{attribute 'linkalways'} 
{attribute 'no_explicit_call' := 'This FB is a CLASS and must be accessed using methods or properties'}
{attribute 'enable_dynamic_creation'}
FUNCTION_BLOCK Node_F_VN_GetPerspectiveTransformation EXTENDS VisionNode
VAR
	aSrcPoints : _TcVnArray4_Point2_REAL;
    aDestPoints : _TcVnArray4_Point2_REAL;
    aTransformationMatrix : _TcVnMatrix3x3_LREAL;
    hrPrev : _HRESULT(S_OK);
	hresult : _HRESULT(S_OK);
END_VAR

METHOD PUBLIC  Clone : I_Node
VAR
	pNode : POINTER TO Node_F_VN_GetPerspectiveTransformation;
END_VAR
pNode := __NEW(Node_F_VN_GetPerspectiveTransformation);
Clone := pNode^;
END_METHOD

METHOD FB_init : BOOL
VAR_INPUT
	bInitRetains : BOOL; // if TRUE, the retain variables are initialized (warm start / cold start)
	bInCopyCode : BOOL;  // if TRUE, the instance afterwards gets moved into the copy code (online change)
END_VAR
AddInput('aSrcPoints', aSrcPoints);
AddInput('aDestPoints', aDestPoints);
AddInput('hrPrev', hrPrev);
AddOutput('aTransformationMatrix', aTransformationMatrix);
AddOutput('hresult',hresult);
END_METHOD

METHOD PROTECTED OnExecute
hresult.Value := F_VN_GetPerspectiveTransformation(
	aSrcPoints := aSrcPoints.Value, 
	aDestPoints := aDestPoints.Value, 
	aTransformationMatrix := aTransformationMatrix.Value, 
	hrPrev := hrPrev.Value);
END_METHOD

METHOD PUBLIC PreExecutionCheck
VAR_INPUT
	Check : I_PreExecutionChecks;
END_VAR
END_METHOD

END_FUNCTION_BLOCK

(* stored: Version 1.1.0.1, ProductVersion 3.1.4024.13
   POU Node_F_VN_GetPerspectiveTransformation: Id {567f5044-920d-0acb-274a-82a5d35ae21f}, SpecialFunc None
   Folder Constructor: Id {fb4ef7d4-23d2-0c39-1ac1-2772d4756ae8}
   Method Clone: Id {65856fbb-4028-0894-01f7-4c9dbae27a33}
   Method FB_init: Id {cd38384d-66e6-001e-27f8-32166a65315e}
   Method OnExecute: Id {ed155c21-c46a-0c11-2c99-78f308492c7d}
   Method PreExecutionCheck: Id {fe563e84-b150-0705-0ef7-55d01b26df10} *)
